// SIMATIC STEP 7 (V5.x) project S7_m2
// CPU: CPU312(1)
// station: P_ADR_BUS
// station: Hardware
// station: SIMATIC 300 Station
// program: S7 Program(1)

SYMBOL_TABLE
"start"	I 0.0	BOOL
"stop"	I 0.1	BOOL
"reset"	I 0.2	BOOL
"box L sensor"	I 0.3	BOOL
"box M sensor"	I 0.4	BOOL
"palletizing box sensor"	I 0.5	BOOL
"pusher box L(back)"	I 0.6	BOOL
"pusher box L(front)"	I 0.7	BOOL
"pusher box M(back)"	I 1.0	BOOL
"pusher box M(front)"	I 1.1	BOOL
"pusher pulletizing front"	I 1.2	BOOL
"pusher pulletizing back"	I 1.3	BOOL
"start(light)"	Q 0.0	BOOL
"stop(light)"	Q 0.1	BOOL
"reset(light)"	Q 0.2	BOOL
"pusher box L"	Q 0.3	BOOL
"pusher box M"	Q 0.4	BOOL
"pusher palletizing box"	Q 0.5	BOOL
"box conveyor"	Q 0.6	BOOL
END_SYMBOL_TABLE

ORGANIZATION_BLOCK OB 1
TITLE = "Main Program Sweep (Cycle)"
VERSION : 0.1
VAR_TEMP
  OB1_EV_CLASS : BYTE ;	//Bits 0-3 = 1 (Coming event), Bits 4-7 = 1 (Event class 1)
  OB1_SCAN_1 : BYTE ;	//1 (Cold restart scan 1 of OB 1), 3 (Scan 2-n of OB 1)
  OB1_PRIORITY : BYTE ;	//Priority of OB Execution
  OB1_OB_NUMBR : BYTE ;	//1 (Organization block 1, OB1)
  OB1_RESERVED_1 : BYTE ;	//Reserved for system
  OB1_RESERVED_2 : BYTE ;	//Reserved for system
  OB1_PREV_CYCLE : INT ;	//Cycle time of previous OB1 scan (milliseconds)
  OB1_MIN_CYCLE : INT ;	//Minimum cycle time of OB1 (milliseconds)
  OB1_MAX_CYCLE : INT ;	//Maximum cycle time of OB1 (milliseconds)
  OB1_DATE_TIME : DATE_AND_TIME ;	//Date and time OB1 started
END_VAR
BEGIN
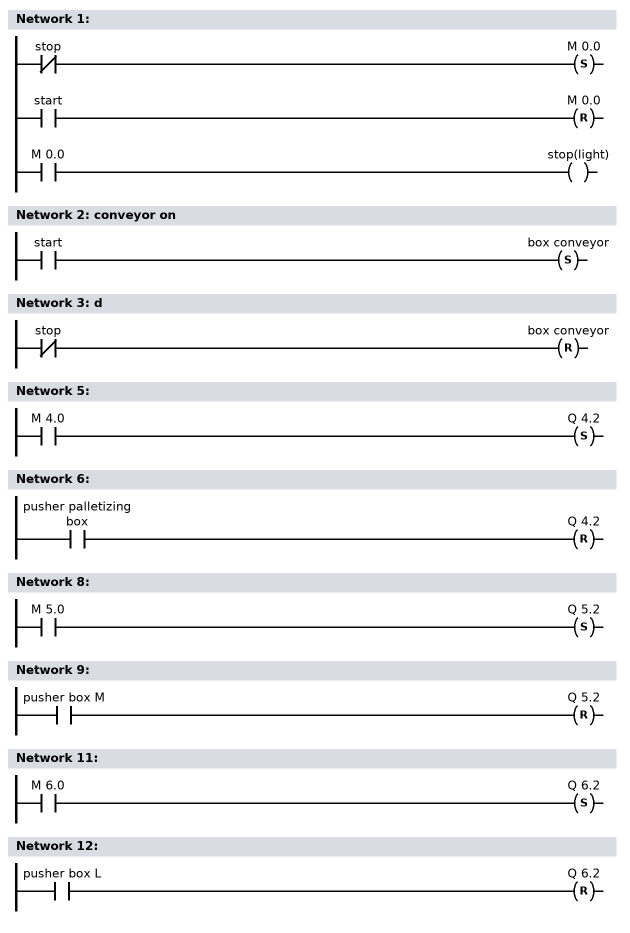
NETWORK
TITLE =
      AN    "stop";
      S     M 0.0;
      A     "start";
      R     M 0.0;
      A     M 0.0;
      =     "stop(light)";
NETWORK
TITLE = conveyor on
      A     "start";
      S     "box conveyor";
NETWORK
TITLE = d
      AN    "stop";
      R     "box conveyor";
NETWORK
TITLE = P
      A(;
      A(;
      A(;
      A(;
      L     128;
      L     ID 30;
      ==D;
      );
      =     M 4.0;
      A     M 4.0;
      CU    C 0;
      BLD   101;
      A     "box conveyor";
      L     C#0;
      S     C 0;
      A(;
      A     "reset";
      JNB   _001;
      L     0;
      T     QD 38;
      SET;
      SAVE;
      CLR;
_001: A     BR;
      );
      R     C 0;
      L     C 0;
      T     MW 30;
      NOP   0;
      A     C 0;
      );
      JNB   _002;
      L     MW 30;
      ITD;
      T     QD 38;
      SET;
      SAVE;
      CLR;
_002: A     BR;
      );
      A(;
      A     M 4.1;
      BLD   100;
      FN    "palletizing box sensor";
      );
      L     S5T#400MS;
      SD    T 1;
      A(;
      O     Q 5.2;
      O     Q 6.2;
      );
      R     T 1;
      NOP   0;
      NOP   0;
      A     T 1;
      );
      L     S5T#1S;
      SF    T 0;
      A     Q 5.2;
      R     T 0;
      NOP   0;
      NOP   0;
      A     T 0;
      =     "pusher palletizing box";
NETWORK
TITLE =
      A     M 4.0;
      S     Q 4.2;
NETWORK
TITLE =
      A     "pusher palletizing box";
      R     Q 4.2;
NETWORK
TITLE = M
      A(;
      A(;
      A(;
      A(;
      L     192;
      L     ID 30;
      ==D;
      );
      =     M 5.0;
      A     M 5.0;
      CU    C 1;
      BLD   101;
      A     "box conveyor";
      L     C#0;
      S     C 1;
      A(;
      A     "reset";
      JNB   _003;
      L     0;
      T     QD 34;
      SET;
      SAVE;
      CLR;
_003: A     BR;
      );
      R     C 1;
      L     C 1;
      T     MW 34;
      NOP   0;
      A     C 1;
      );
      JNB   _004;
      L     MW 34;
      ITD;
      T     QD 34;
      SET;
      SAVE;
      CLR;
_004: A     BR;
      );
      A(;
      A     M 5.1;
      BLD   100;
      FN    "box M sensor";
      );
      L     S5T#400MS;
      SD    T 2;
      A(;
      O     Q 4.2;
      O     Q 6.2;
      );
      R     T 2;
      NOP   0;
      NOP   0;
      A     T 2;
      );
      L     S5T#1S;
      SF    T 3;
      A     Q 4.2;
      R     T 3;
      NOP   0;
      NOP   0;
      A     T 3;
      =     "pusher box M";
NETWORK
TITLE =
      A     M 5.0;
      S     Q 5.2;
NETWORK
TITLE =
      A     "pusher box M";
      R     Q 5.2;
NETWORK
TITLE = L
      A(;
      A(;
      A(;
      A(;
      A(;
      L     224;
      L     ID 30;
      ==D;
      );
      =     M 6.0;
      A     M 6.0;
      S     M 6.0;
      A     "pusher box L";
      R     M 6.0;
      A     M 6.0;
      );
      CU    C 2;
      BLD   101;
      A     "box conveyor";
      L     C#0;
      S     C 2;
      A(;
      A     "reset";
      JNB   _005;
      L     0;
      T     QD 30;
      SET;
      SAVE;
      CLR;
_005: A     BR;
      );
      R     C 2;
      L     C 2;
      T     MW 38;
      NOP   0;
      A     C 2;
      );
      JNB   _006;
      L     MW 38;
      ITD;
      T     QD 30;
      SET;
      SAVE;
      CLR;
_006: A     BR;
      );
      A(;
      A     M 6.1;
      BLD   100;
      FN    "box L sensor";
      );
      L     S5T#400MS;
      SD    T 4;
      A(;
      O     Q 4.2;
      O     Q 5.2;
      );
      R     T 4;
      NOP   0;
      NOP   0;
      A     T 4;
      );
      L     S5T#1S;
      SF    T 5;
      NOP   0;
      NOP   0;
      NOP   0;
      A     T 5;
      =     "pusher box L";
NETWORK
TITLE =
      A     M 6.0;
      S     Q 6.2;
NETWORK
TITLE =
      A     "pusher box L";
      R     Q 6.2;
END_ORGANIZATION_BLOCK
